PROGRAM MAIN
VAR
END_VAR

END_PROGRAM

(* stored: Version 1.1.0.1
   POU MAIN: Id {9373ef9e-5e95-4b75-81c2-b0e4a1795889} *)
